FUNCTION_BLOCK Stagesss22 (* Template for a Basic Function Block Type *)
  (* Standard: 61499-2 *)
  (* Version 1.0, 2021-06-20, HP *)
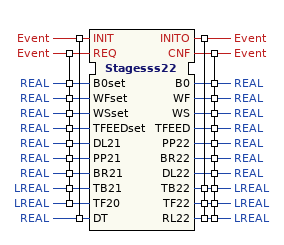
  EVENT_INPUT
    INIT WITH DT; (* Initialization Request *)
    REQ WITH WFset, WSset, TFEEDset, DL21, PP21, BR21, TB21, TF20, B0set; (* Normal Execution Request *)
  END_EVENT
  EVENT_OUTPUT
    INITO WITH TB22, TF22, RL22; (* Initialization Confirm *)
    CNF WITH TB22, DL22, TF22, BR22, PP22, TFEED, WF, WS, RL22, B0; (* Execution Confirmation *)
  END_EVENT
  VAR_INPUT
    B0set : REAL;
    WFset : REAL;
    WSset : REAL;
    TFEEDset : REAL;
    DL21 : REAL;
    PP21 : REAL;
    BR21 : REAL;
    TB21 : LREAL;
    TF20 : LREAL;
    DT : REAL;
  END_VAR
  VAR_OUTPUT
    B0 : REAL;
    WF : REAL;
    WS : REAL;
    TFEED : REAL;
    PP22 : REAL;
    BR22 : REAL;
    DL22 : REAL;
    TB22 : LREAL;
    TF22 : LREAL;
    RL22 : LREAL;
  END_VAR
  VAR
    AB : REAL; (* internal variabel *)
    UU : REAL;
    REJ : REAL;
    WMK : REAL;
    TREF : REAL;
    AD : REAL;
    AHC : REAL;
    AHR : REAL;
    AS : REAL;
    REC : REAL;
    WN : REAL;
    WN_1 : REAL;
    XKN : REAL;
    C1 : REAL;
    HS : REAL;
    G : REAL;
    W1 : REAL;
    TFREC : REAL;
    TS : REAL;
    DTS : REAL;
    TF22_last : REAL;
    RL22_last : REAL;
    TB22_last : REAL;
    USS : REAL;
    RHOB : REAL;
    CPB : REAL;
    CPF : REAL;
    FMW : REAL;
    HLV : REAL;
    HV : REAL;
    BPR : REAL;
    FMC : REAL;
    U : REAL;
    A : REAL;
    B : REAL;
    C : REAL;
    D1 : REAL;
    d : REAL;
    a : REAL;
    A1 : REAL;
    A2 : REAL;
    A3 : REAL;
    A4 : REAL;
    A5 : REAL;
    A6 : REAL;
    p : REAL;
    q : REAL;
    TC : REAL;
    PC : REAL;
    DTB22 : REAL;
    DEN22 : REAL;
    DH22 : REAL;
    DP22 : REAL;
    DPDH22 : REAL;
    DT22 : REAL;
    m : REAL;
    n : REAL;
    VR22 : REAL;
    DELTA22 : REAL;
    DELTA44 : REAL;
    DELTA66 : REAL;
    DELTA22_last : REAL;
    DELTA44_last : REAL;
    DELTA66_last : REAL;
  END_VAR
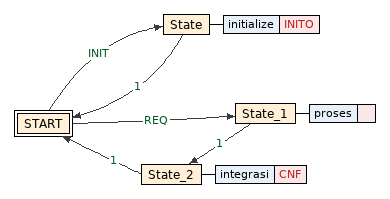
  EC_STATES
    START; (* Initial State *)
    State : initialize -> INITO;
    State_1 : proses;
    State_2 : integrasi -> CNF;
  END_STATES
  EC_TRANSITIONS
    START TO State := INIT;
    State TO START := 1;
    START TO State_1 := REQ;
    State_1 TO State_2 := 1;
    State_2 TO START := 1;
  END_TRANSITIONS
  ALGORITHM initialize IN ST: (* Initialization algorithm *)
TREF :=273.15;
AB :=57.2727;
AHC :=4069.2;
AHR :=2639.7;
AS :=3225.7;
REC :=0.0;
//TF2:=TF2;

//TFEED :=TFEED1+TREF;
 //TS:=TS1+TREF;
WN :=3.0;
XKN :=0.68;
HS:=0.11;
G :=9.81;
W1 :=0.50;

RL22 := 0.556817361925019;
TB22 := 314.548634310388;
TF22 := 310.669094657679;
TF20 := 314.769851417199;


RL22_last :=RL22;
TB22_last :=TB22;
TF22_last :=TF22;
  END_ALGORITHM
  ALGORITHM proses IN ST: (* kalkulasi *)
B0 :=B0set;
WS :=WSset;
WF:=WFset;
TFEED:=TFEEDset;
TFEED:=TFEEDset;
UU := TFEEDset;
U :=UU;

REC :=0.0;
REJ:=95.35;
WMK:=WF-REJ-REC;

USS :=49.767;
C1 :=0.625;
RHOB :=1032.4; //maassa jenis brine
CPB :=1.00; //heatcapacity Brine
CPF :=1.00; //heat capacity feed
FMW :=23654.0;
HLV :=563.7959;
HV :=625.1971;
BPR :=2.192;
FMC :=34736.09;
//U :=UU; //feed temp



///  Calculate the physical properties

//A :=3.2437814;
//B :=5.86826*0.001;
//C :=1.1702379*0.00000001;
//D1 :=2.1878462*0.001;
//TC :=647.27;
//PC :=218.167;


A1 :=3.2437814;
A2:=5.86826*0.001;
A3:=1.1702379*0.00000001;
A4 :=2.1878462*0.001;
A5 :=647.27;
A6 :=218.167;

DTB22 :=A5-TB22;
DEN22 :=(A1+A2*DTB22+A3*DTB22*DTB22*DTB22)/(1+A4*DTB22)*DTB22/TB22;
p:=DEN22;
q:=10.0;
PP22 :=A6/(EXPT(q, p));

// calculate the brine flow rates
DP22:=PP21-PP22;
DH22:=RL22-C1*HS;
DPDH22 :=DP22*101000+G*RHOB*DH22;
m:=DPDH22*RHOB;
n:=0.5;
BR22 :=W1*XKN*RL22*(EXPT(m, n));
BR22 :=BR22*60.0/1000.0;

// calculate the vapor flow rates

DT22 :=TB22-BPR/1.8-(TFEED+TF22)*0.5;
VR22:=U*AHR*DT22/HLV/1000.0;
DL22 :=DL21+VR22;


//// state equation
DELTA22 :=(BR21-BR22-VR22-B0+WMK)*1000.0/RHOB/AB;
DELTA44 :=((BR21*CPB*(TB21-TB22))+(WMK*CPB*(TF20-TB22))-VR22*(HV-CPB*(TB22-TREF)))*1000.0/AB/RHOB/CPB/RL22;
DELTA66 :=(WF*CPF*(TFEED-TF22)*1000+(U*AHR*DT22))/FMW/CPF;
  END_ALGORITHM
  ALGORITHM integrasi IN ST: (* new algorithm *)
B0:=B0set;
WF :=WFset;
WS :=WSset;
TFEED:=TFEEDset;
//integrasi
RL22 := (DELTA22 + DELTA22_last)*0.5*DT + RL22_last;
DELTA22_last :=DELTA22 ;
RL22_last :=RL22;

TB22:= (DELTA44 + DELTA44_last)*0.5*DT + TB22_last;
DELTA44_last :=DELTA44 ;
TB22_last:=TB22;

TF22 := (DELTA66 + DELTA66_last)*0.5*DT + TF22_last;
DELTA66_last :=DELTA66 ;
TF22_last :=TF22;
  END_ALGORITHM
END_FUNCTION_BLOCK
